{attribute 'hide'}
PROGRAM MAIN
VAR
	state : (IDLE, FIND_FILES, USE_FILES, CLEANUP, DONE) := IDLE;
	fileFinder : FileFinder;
	fileCollection : FileSystemEntryCollection;
	searchPath : FilePath := 'C:\temp\integration\';
	fileSystemEntry : I_FileSystemEntry;
	disposable : I_Disposable;
	path : FilePath;
	append : BOOL;
	index : INT;
	check : BOOL;
END_VAR

General_TestSuite();
FileSystem_TestSuite();

TcUnit.RUN();

// find files in supplied initial folder & sub-folders and populate a collection.
CASE state OF 
	
	IDLE : //
	
	FIND_FILES:
		IF (fileFinder.Find(searchPath, '*.tcgraph', fileCollection, append)) THEN
			state := USE_FILES;
		END_IF
	
	USE_FILES:
		state := CLEANUP;
		
	CLEANUP:
		state := DONE;
		
	DONE:
		;
			
END_CASE

IF check THEN
	check := FALSE;
	path := fileCollection.GetByIndex(26).Path;
END_IF

END_PROGRAM

(* stored: Version 1.1.0.1, ProductVersion 3.1.4024.9
   POU MAIN: Id {ec38523b-9156-4770-8e81-c6221898da8f}, SpecialFunc None *)
